KUKA KRL data list: Station1.dat

&ACCESS RV
&REL 2
DEFDAT  Station1 PUBLIC

ENDDAT
